// TIA Portal V17 export
// export: Created 2026-07-18T05:18:17.1039229Z, ExportSetting WithDefaults, DisplayName Totally Integrated Automation Portal, DisplayVersion V17 Update 7, DisplayName TIA Portal Openness, DisplayVersion V17 Update 7, DisplayName TIA Portal Version Control Interface, DisplayVersion V17, DisplayName SINAMICS Startdrive Advanced, DisplayVersion V17 SP2, DisplayName SINAMICS Startdrive G110M, G120, G120C, G120D, G120P, G115D, DisplayVersion V17 SP2, DisplayName SINAMICS Startdrive G130, G150, S120, S150, SINAMICS MV, S210, DisplayVersion V17 SP2, DisplayName STEP 7 Professional, DisplayVersion V17 Update 7, DisplayName STEP 7 Safety, DisplayVersion V17 Update 6, DisplayName WinCC Advanced, DisplayVersion V17 Update 7
ORGANIZATION_BLOCK "Main"   // OB1, LAD, ProgramCycle
TITLE = "Main Program Sweep (Cycle)"
{ S7_Optimized_Access := 'TRUE' }
VERSION : 0.1
// stored: AutoNumber true, IsIECCheckEnabled false, SetENOAutomatically false
   VAR_INPUT
      Initial_Call : Bool;   // Initial call of this OB
      Remanence : Bool;   // =True, if remanent data are available
   END_VAR
BEGIN

REGION Network 1
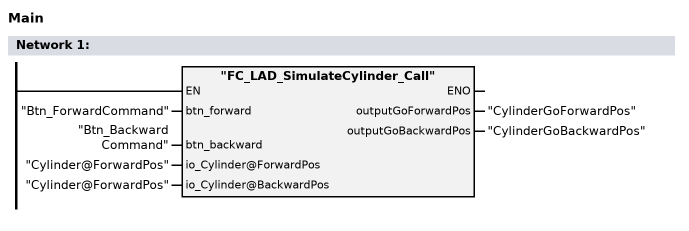
   RUNG wire#powerrail
      "FC_LAD_SimulateCylinder_Call"(btn_forward := "Btn_ForwardCommand", btn_backward := "Btn_BackwardCommand", "io_Cylinder@ForwardPos" := "Cylinder@ForwardPos", "io_Cylinder@BackwardPos" := "Cylinder@ForwardPos", outputGoForwardPos => "CylinderGoForwardPos", outputGoBackwardPos => "CylinderGoBackwardPos")
   END_RUNG
   // the same network as SCL:
   "FC_LAD_SimulateCylinder_Call"(btn_forward := "Btn_ForwardCommand",
                           btn_backward := "Btn_BackwardCommand",
                           "io_Cylinder@ForwardPos" := "Cylinder@ForwardPos",
                           "io_Cylinder@BackwardPos" := "Cylinder@ForwardPos",
                           outputGoForwardPos => "CylinderGoForwardPos",
                           outputGoBackwardPos => "CylinderGoBackwardPos");
END_REGION
END_ORGANIZATION_BLOCK
